PROGRAM PRG_Cycle
VAR	
Status : INT := 0;
bHomingDone: BOOL;
bCycleDone: BOOL;
SFCReset : BOOL;
END_VAR

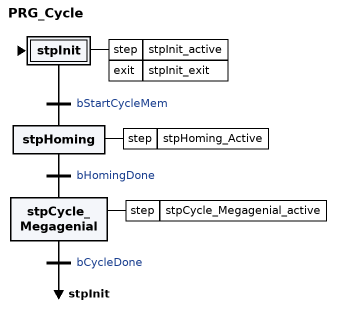
INITIAL_STEP stpInit:
    stpInit_active(N);  // step action
    stpInit_exit(P0);  // exit action
END_STEP
TRANSITION FROM stpInit TO stpHoming
    := bStartCycleMem;
END_TRANSITION
STEP stpHoming:
    stpHoming_Active(N);  // step action
END_STEP
TRANSITION FROM stpHoming TO stpCycle_Megagenial
    := bHomingDone;
END_TRANSITION
STEP stpCycle_Megagenial:
    stpCycle_Megagenial_active(N);  // step action
END_STEP
TRANSITION FROM stpCycle_Megagenial TO stpInit
    := bCycleDone;
END_TRANSITION

ACTION _astpCatch_Rail1_active:
Status := F_IssueActuatorCommand(sDevice := 'R1_Chariot', bArg := TRUE);

CASE Status OF
	1: Result := 0;
	
	0: //Continue
	
	-1: bStopCycleMem := FALSE;
		bStartCycleMem := FALSE;
		bHomingDone := FALSE;
		bCycleDone := FALSE;
		Result := 0;
		SFCReset := TRUE;
END_CASE
END_ACTION

ACTION _astpCatch_Rail1_entry:
Status := 0;
END_ACTION

ACTION _astpCatch_Rail2_active:
Status := F_IssueActuatorCommand(sDevice := 'R2_Chariot', bArg := TRUE);

CASE Status OF
	1: Result := 0;
	
	0: //Continue
	
	-1: bStopCycleMem := FALSE;
		bStartCycleMem := FALSE;
		bHomingDone := FALSE;
		bCycleDone := FALSE;
		Result := 0;
		SFCReset := TRUE;
END_CASE
END_ACTION

ACTION _astpCatch_Rail2_entry:
Status := 0;
END_ACTION

ACTION _astpCatch_Rail3_active:
Status := F_IssueActuatorCommand(sDevice := 'R3_Chariot', bArg := TRUE);

CASE Status OF
	1: Result := 0;
	
	0: //Continue
	
	-1: bStopCycleMem := FALSE;
		bStartCycleMem := FALSE;
		bHomingDone := FALSE;
		bCycleDone := FALSE;
		Result := 0;
		SFCReset := TRUE;
END_CASE
END_ACTION

ACTION _astpCatch_Rail3_entry:
Status := 0;
END_ACTION

ACTION _astpCatch_Rail4_active:
Status := F_IssueActuatorCommand(sDevice := 'R4_Chariot', bArg := TRUE);

CASE Status OF
	1: Result := 0;
	
	0: //Continue
	
	-1: bStopCycleMem := FALSE;
		bStartCycleMem := FALSE;
		bHomingDone := FALSE;
		bCycleDone := FALSE;
		Result := 0;
		SFCReset := TRUE;
END_CASE
END_ACTION

ACTION _astpCatch_Rail4_entry:
Status := 0;
END_ACTION

ACTION _astpCatchPickUp_Rail3_active:
Status := F_IssueActuatorCommand(sDevice := 'R3_Chariot', bArg := TRUE);

CASE Status OF
	1: Result := 0;
	
	0: //Contionue
	
	-1: bStopCycleMem := FALSE;
		bStartCycleMem := FALSE;
		bHomingDone := FALSE;
		bCycleDone := FALSE;
		Result := 0;
		SFCReset := TRUE;
END_CASE
END_ACTION

ACTION _astpCatchPickUp_Rail3_entry:
Status := 0;
END_ACTION

ACTION _astpDrop_Gui1_active:
Status := F_IssueActuatorCommand(sDevice := 'R3_HeatExCoupola', bArg := FALSE);

CASE Status OF
	1: Result := 0;
	
	0: //Continue
	
	-1: bStopCycleMem := FALSE;
		bStartCycleMem := FALSE;
		bHomingDone := FALSE;
		bCycleDone := FALSE;
		Result := 0;
		SFCReset := TRUE;
END_CASE
END_ACTION

ACTION _astpDrop_Gui1_entry:
Status := 0;
END_ACTION

ACTION _astpDrop_Rail1_entry:
Status := 0;
END_ACTION

ACTION _astpDrop_Rail2_active:
Status := F_IssueActuatorCommand(sDevice := 'R2_Chariot', bArg := FALSE);

CASE Status OF
	1: Result := 0;
	
	0: //Continue
	
	-1: bStopCycleMem := FALSE;
		bStartCycleMem := FALSE;
		bHomingDone := FALSE;
		bCycleDone := FALSE;
		Result := 0;
		SFCReset := TRUE;
END_CASE
END_ACTION

ACTION _astpDrop_Rail2_entry:
Status := 0;
END_ACTION

ACTION _astpDrop_Rail3_active:
Status := F_IssueActuatorCommand(sDevice := 'R3_Chariot', bArg := FALSE);

CASE Status OF
	1: Result := 0;
	
	0: //Continue
	
	-1: bStopCycleMem := FALSE;
		bStartCycleMem := FALSE;
		bHomingDone := FALSE;
		bCycleDone := FALSE;
		Result := 0;
		SFCReset := TRUE;
END_CASE
END_ACTION

ACTION _astpDrop_Rail3_entry:
Status := 0;
END_ACTION

ACTION _astpDrop_Rail4_active_1:
Status := F_IssueActuatorCommand(sDevice := 'R4_Chariot', bArg := FALSE);

CASE Status OF
	1: Result := 0;
	
	0: //Continue
	
	-1: bStopCycleMem := FALSE;
		bStartCycleMem := FALSE;
		bHomingDone := FALSE;
		bCycleDone := FALSE;
		Result := 0;
		SFCReset := TRUE;
END_CASE
END_ACTION

ACTION _astpDrop_Rail4_entry:
Status := 0;
END_ACTION

ACTION _astpDropMoveFinal_Rail3_active:
Status := F_IssueActuatorCommand(sDevice := 'R3_Chariot', bArg := FALSE);

CASE Status OF
	1: Result := 0;
	
	0: //Contionue
	
	-1: bStopCycleMem := FALSE;
		bStartCycleMem := FALSE;
		bHomingDone := FALSE;
		bCycleDone := FALSE;
		Result := 0;
		SFCReset := TRUE;
END_CASE
END_ACTION

ACTION _astpDropMoveFinal_Rail3_entry:
Status := 0;
END_ACTION

ACTION _astpEnd_active:
IF bStopCycleMem THEN
	bStartCycleMem := FALSE;
	bStopCycleMem := FALSE;
	bHomingDone := FALSE;
END_IF

bHomingDone := FALSE;
bCycleDone := TRUE;
END_ACTION

ACTION _astpExtend_Pous2_active:
Status := F_IssueActuatorCommand(sDevice := 'R3_Compressor', bArg := TRUE);

CASE Status OF
	1: Result := 0;
	
	0: //Continue
	
	-1: bStopCycleMem := FALSE;
		bStartCycleMem := FALSE;
		bHomingDone := FALSE;
		bCycleDone := FALSE;
		Result := 0;
		SFCReset := TRUE;
END_CASE
END_ACTION

ACTION _astpExtend_Pous2_entry:
Status := 0;
END_ACTION

ACTION _astpHoming_Gui1_active:
Status := F_IssueActuatorCommand(sDevice := 'R3_HeatExCoupola', bArg := TRUE);

CASE Status OF
	1: Result := 0;
	
	0: //Continue
	
	-1: bStopCycleMem := FALSE;
		bStartCycleMem := FALSE;
		bHomingDone := FALSE;
		bCycleDone := FALSE;
		Result := 0;
		SFCReset := TRUE;
END_CASE
END_ACTION

ACTION _astpHoming_Gui1_entry:
Status := 0;
END_ACTION

ACTION _astpHoming_Gui2_active:
Status := F_IssueActuatorCommand(sDevice := 'R3_RegenCoupola', bArg := TRUE);

CASE Status OF
	1: Result := 0;
	
	0: //Continue
	
	-1: bStopCycleMem := FALSE;
		bStartCycleMem := FALSE;
		bHomingDone := FALSE;
		bCycleDone := FALSE;
		Result := 0;
		SFCReset := TRUE;
END_CASE
END_ACTION

ACTION _astpHoming_Gui2_entry:
Status := 0;
END_ACTION

ACTION _astpHoming_Pous1_active:
Status := F_IssueActuatorCommand(sDevice := 'R1_Compressor', bArg := FALSE);

CASE Status OF
	1: Result := 0;
	
	0: //Continue
	
	-1: bStopCycleMem := FALSE;
		bStartCycleMem := FALSE;
		bHomingDone := FALSE;
		bCycleDone := FALSE;
		Result := 0;
		SFCReset := TRUE;
END_CASE
END_ACTION

ACTION _astpHoming_Pous1_entry:
Status := 0;
END_ACTION

ACTION _astpHoming_Pous2_active:
Status := F_IssueActuatorCommand(sDevice := 'R3_Compressor', bArg := FALSE);

CASE Status OF
	1: Result := 0;
	   bHomingDone := TRUE;
	
	0: //Continue
	
	-1: bStopCycleMem := FALSE;
		bStartCycleMem := FALSE;
		bHomingDone := FALSE;
		bCycleDone := FALSE;
		Result := 0;
		SFCReset := TRUE;
END_CASE
END_ACTION

ACTION _astpHoming_Pous2_entry:
Status := 0;
END_ACTION

ACTION _astpHoming_Rail1_entry:
Status := 0;
END_ACTION

ACTION _astpHoming_Rail2_entry:
Status := 0;
END_ACTION

ACTION _astpHoming_Rail3_entry:
Status := 0;
END_ACTION

ACTION _astpHoming_Rail4_entry:
Status := 0;
END_ACTION

ACTION _astpHoming_Tri1_active:
Status := F_IssueActuatorCommand(sDevice := 'R1_Chariot', bArg := FALSE);

CASE Status OF
	1: Result := 0;
	
	0: //Continue
	
	-1: bStopCycleMem := FALSE;
		bStartCycleMem := FALSE;
		bHomingDone := FALSE;
		bCycleDone := FALSE;
		Result := 0;
		SFCReset := TRUE;
END_CASE
END_ACTION

ACTION _astpHoming_Tri1_entry:
Status := 0;
END_ACTION

ACTION _astpHoming_Tri2_active:
IF bStopCycleMem THEN
	sRequestedActuator := 'none';
	CancelMove := TRUE;
ELSIF NOT bStopCycleMem THEN
	Status := F_IssueActuatorCommand(sDevice := 'R2_Chariot', bArg := FALSE);
END_IF

IF Status = 1 THEN
	Result := 0;
END_IF
END_ACTION

ACTION _astpHoming_Tri2_active_1:
Status := F_IssueActuatorCommand(sDevice := 'R2_Chariot', bArg := FALSE);

CASE Status OF
	1: Result := 0;
	
	0: //Continue
	
	-1: bStopCycleMem := FALSE;
		bStartCycleMem := FALSE;
		bHomingDone := FALSE;
		bCycleDone := FALSE;
		Result := 0;
		SFCReset := TRUE;
END_CASE
END_ACTION

ACTION _astpHoming_Tri2_entry:
Status := 0;
END_ACTION

ACTION _astpHoming_Tri2_entry_1:
Status := 0;
END_ACTION

ACTION _astpHoming_Tri3_active:
Status := F_IssueActuatorCommand(sDevice := 'R3_Chariot', bArg := FALSE);

CASE Status OF
	1: Result := 0;
	
	0: //Continue
	
	-1: bStopCycleMem := FALSE;
		bStartCycleMem := FALSE;
		bHomingDone := FALSE;
		bCycleDone := FALSE;
		Result := 0;
		SFCReset := TRUE;
END_CASE
END_ACTION

ACTION _astpHoming_Tri3_entry:
Status := 0;
END_ACTION

ACTION _astpHoming_Tri4_active:
Status := F_IssueActuatorCommand(sDevice := 'R4_Chariot', bArg := FALSE);

CASE Status OF
	1: Result := 0;
	
	0: //Continue
	
	-1: bStopCycleMem := FALSE;
		bStartCycleMem := FALSE;
		bHomingDone := FALSE;
		bCycleDone := FALSE;
		Result := 0;
		SFCReset := TRUE;
END_CASE
END_ACTION

ACTION _astpHoming_Tri4_entry:
Status := 0;
END_ACTION

ACTION _astpInit_Cycle_Megagenial_active:

END_ACTION

ACTION _astpInit_Homing_active:

END_ACTION

ACTION _astpMoveBw_Rail1_active:
Status := F_IssueActuatorCommand(sDevice := 'R1_Motor', bArg := FALSE, bHasPosition := TRUE, nPosition:= 6, fVelocity := Mot_LoadedVel);
	
CASE Status OF
	1: Result := 0;
	
	0: //Continue
	
	-1: bStopCycleMem := FALSE;
		bStartCycleMem := FALSE;
		bHomingDone := FALSE;
		bCycleDone := FALSE;
		Result := 0;
		SFCReset := TRUE;
END_CASE
END_ACTION

ACTION _astpMoveBw_Rail1_entry:
Status := 0;
END_ACTION

ACTION _astpMoveBw_Rail2_active:
Status := F_IssueActuatorCommand(sDevice := 'R2_Motor', bArg := FALSE, bHasPosition := TRUE, nPosition:= 6, fVelocity := Mot_LoadedVel);

CASE Status OF
	1: Result := 0;
	
	0: //Continue
	
	-1: bStopCycleMem := FALSE;
		bStartCycleMem := FALSE;
		bHomingDone := FALSE;
		bCycleDone := FALSE;
		Result := 0;
		SFCReset := TRUE;
END_CASE
END_ACTION

ACTION _astpMoveBw_Rail2_entry:
Status := 0;
END_ACTION

ACTION _astpMoveBw_Rail3_active:
Status := F_IssueActuatorCommand(sDevice := 'R3_Motor', bArg := FALSE, bHasPosition := TRUE, nPosition:= 6, fVelocity := Mot_LoadedVel);
	
CASE Status OF
	1: Result := 0;
	
	0: //Continue
	
	-1: bStopCycleMem := FALSE;
		bStartCycleMem := FALSE;
		bHomingDone := FALSE;
		bCycleDone := FALSE;
		Result := 0;
		SFCReset := TRUE;
END_CASE
END_ACTION

ACTION _astpMoveBw_Rail3_entry:
Status := 0;
END_ACTION

ACTION _astpMoveBw_Rail4_active:
Status := F_IssueActuatorCommand(sDevice := 'R4_Motor', bArg := FALSE, bHasPosition := TRUE, nPosition:= 9, fVelocity := Mot_LoadedVel);

CASE Status OF
	1: Result := 0;
	
	0: //Continue
	
	-1: bStopCycleMem := FALSE;
		bStartCycleMem := FALSE;
		bHomingDone := FALSE;
		bCycleDone := FALSE;
		Result := 0;
		SFCReset := TRUE;
END_CASE
END_ACTION

ACTION _astpMoveBw_Rail4_entry:
Status := 0;
END_ACTION

ACTION _astpMoveFinal_Rail3_active:
Status := F_IssueActuatorCommand(sDevice := 'R3_Motor', bArg := FALSE, bHasPosition := TRUE, nPosition:= 6, fVelocity := Mot_UnloadedVel);

CASE Status OF
	1: Result := 0;
	
	0: //Contionue
	
	-1: bStopCycleMem := FALSE;
		bStartCycleMem := FALSE;
		bHomingDone := FALSE;
		bCycleDone := FALSE;
		Result := 0;
		SFCReset := TRUE;
END_CASE
END_ACTION

ACTION _astpMoveFinal_Rail3_entry:
Status := 0;
END_ACTION

ACTION _astpMoveFw_Rail1_active:
Status := F_IssueActuatorCommand(sDevice := 'R1_Motor', bArg := FALSE, bHasPosition := TRUE, nPosition:= 1290, fVelocity := Mot_UnloadedVel);

CASE Status OF
	1: Result := 0;
	
	0: //Continue
	
	-1: bStopCycleMem := FALSE;
		bStartCycleMem := FALSE;
		bHomingDone := FALSE;
		bCycleDone := FALSE;
		Result := 0;
		SFCReset := TRUE;
END_CASE
END_ACTION

ACTION _astpMoveFw_Rail1_entry:
Status := 0;
END_ACTION

ACTION _astpMoveFw_Rail2_active:
Status := F_IssueActuatorCommand(sDevice := 'R2_Motor', bArg := FALSE, bHasPosition := TRUE, nPosition:= 980, fVelocity := Mot_UnloadedVel);

CASE Status OF
	1: Result := 0;
	
	0: //Continue
	
	-1: bStopCycleMem := FALSE;
		bStartCycleMem := FALSE;
		bHomingDone := FALSE;
		bCycleDone := FALSE;
		Result := 0;
		SFCReset := TRUE;
END_CASE
END_ACTION

ACTION _astpMoveFw_Rail2_entry:
Status := 0;
END_ACTION

ACTION _astpMoveFw_Rail3_active:
Status := F_IssueActuatorCommand(sDevice := 'R3_Motor', bArg := FALSE, bHasPosition := TRUE, nPosition:= 1290, fVelocity := Mot_UnloadedVel);

CASE Status OF
	1: Result := 0;
	
	0: //Contionue
	
	-1: bStopCycleMem := FALSE;
		bStartCycleMem := FALSE;
		bHomingDone := FALSE;
		bCycleDone := FALSE;
		Result := 0;
		SFCReset := TRUE;
END_CASE
END_ACTION

ACTION _astpMoveFw_Rail3_entry:
Status := 0;
END_ACTION

ACTION _astpMoveFw_Rail4_active:
Status := F_IssueActuatorCommand(sDevice := 'R4_Motor', bArg := FALSE, bHasPosition := TRUE, nPosition:= 980, fVelocity := Mot_UnloadedVel);

CASE Status OF
	1: Result := 0;
	
	0: //Continue
	
	-1: bStopCycleMem := FALSE;
		bStartCycleMem := FALSE;
		bHomingDone := FALSE;
		bCycleDone := FALSE;
		Result := 0;
		SFCReset := TRUE;
END_CASE
END_ACTION

ACTION _astpMoveFw_Rail4_entry:
Status := 0;
END_ACTION

ACTION _astpMovePickUp_Rail3_active:
Status := F_IssueActuatorCommand(sDevice := 'R3_Motor', bArg := FALSE, bHasPosition := TRUE, nPosition:= 150, fVelocity := Mot_UnloadedVel);

CASE Status OF
	1: Result := 0;
	
	0: //Contionue
	
	-1: bStopCycleMem := FALSE;
		bStartCycleMem := FALSE;
		bHomingDone := FALSE;
		bCycleDone := FALSE;
		Result := 0;
		SFCReset := TRUE;
END_CASE
END_ACTION

ACTION _astpMovePickUp_Rail3_entry:
Status := 0;
END_ACTION

ACTION _astpPivotIn_active:
Status := F_IssueActuatorCommand(sDevice := 'R1_Sensor', bArg := FALSE);

CASE Status OF
	1: Result := 0;
	
	0: //Continue
	
	-1: bStopCycleMem := FALSE;
		bStartCycleMem := FALSE;
		bHomingDone := FALSE;
		bCycleDone := FALSE;
		Result := 0;
		SFCReset := TRUE;
END_CASE
END_ACTION

ACTION _astpPivotIn_entry:
Status := 0;
END_ACTION

ACTION _astpPivotOut_active:
Status := F_IssueActuatorCommand(sDevice := 'R1_Sensor', bArg := TRUE);

CASE Status OF
	1: Result := 0;
	
	0: //Continue
	
	-1: bStopCycleMem := FALSE;
		bStartCycleMem := FALSE;
		bHomingDone := FALSE;
		bCycleDone := FALSE;
		Result := 0;
		SFCReset := TRUE;
END_CASE
END_ACTION

ACTION _astpPivotOut_entry:
Status := 0;
END_ACTION

ACTION _astpRetract_Gui1_active:
Status := F_IssueActuatorCommand(sDevice := 'R3_HeatExCoupola', bArg := TRUE);

CASE Status OF
	1: Result := 0;
	
	0: //Contionue
	
	-1: bStopCycleMem := FALSE;
		bStartCycleMem := FALSE;
		bHomingDone := FALSE;
		bCycleDone := FALSE;
		Result := 0;
		SFCReset := TRUE;
END_CASE
END_ACTION

ACTION _astpRetract_Gui1_entry:
Status := 0;
END_ACTION

ACTION _astpRetract_Pous2_active:
Status := F_IssueActuatorCommand(sDevice := 'R3_Compressor', bArg := FALSE);

CASE Status OF
	1: Result := 0;
	
	0: //Continue
	
	-1: bStopCycleMem := FALSE;
		bStartCycleMem := FALSE;
		bHomingDone := FALSE;
		bCycleDone := FALSE;
		Result := 0;
		SFCReset := TRUE;
END_CASE
END_ACTION

ACTION _astpRetract_Pous2_entry:
Status := 0;
END_ACTION

ACTION stpCycle_Megagenial_active:
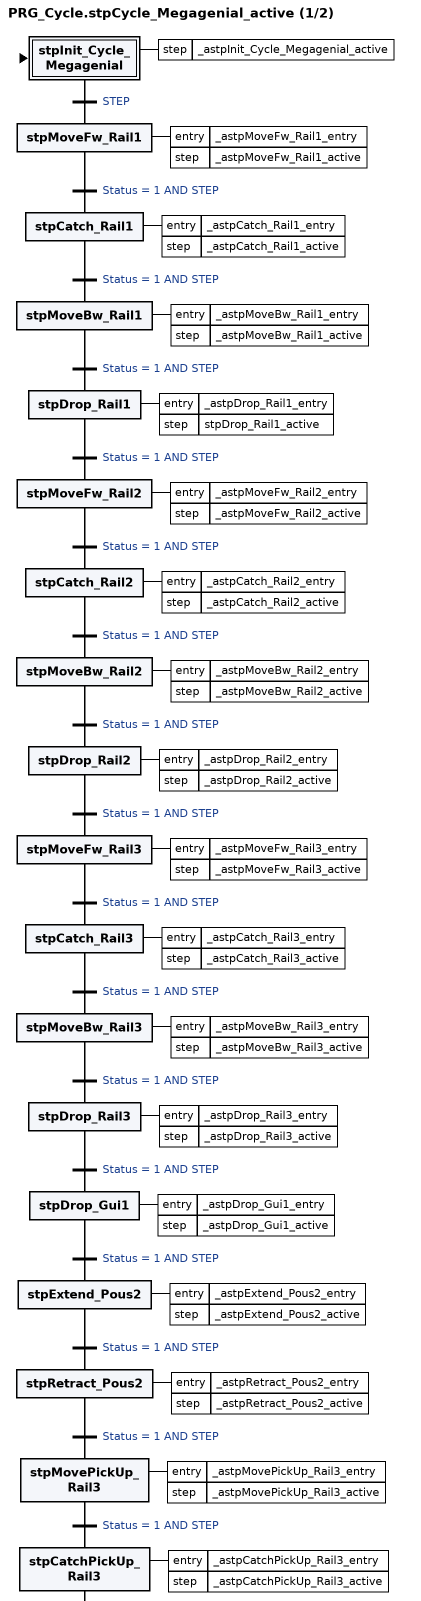
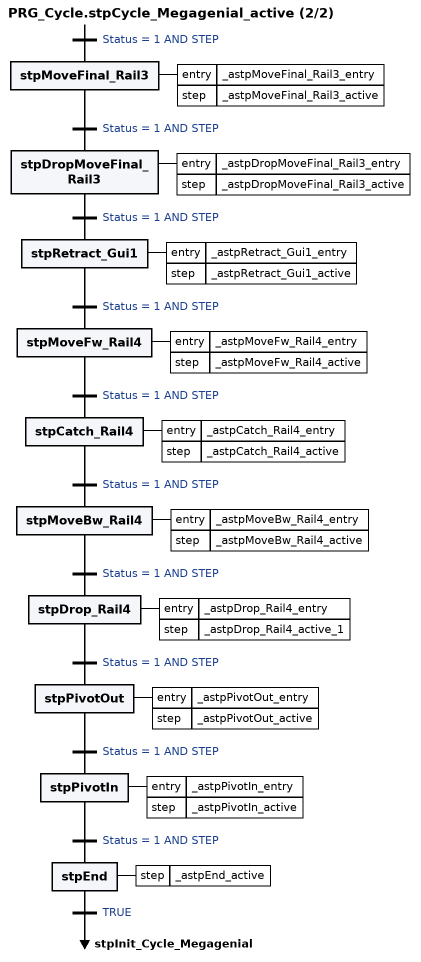
INITIAL_STEP stpInit_Cycle_Megagenial:
    _astpInit_Cycle_Megagenial_active(N);  // step action
END_STEP
TRANSITION FROM stpInit_Cycle_Megagenial TO stpMoveFw_Rail1
    := STEP;
END_TRANSITION
STEP stpMoveFw_Rail1:
    _astpMoveFw_Rail1_entry(P1);  // entry action
    _astpMoveFw_Rail1_active(N);  // step action
END_STEP
TRANSITION FROM stpMoveFw_Rail1 TO stpCatch_Rail1
    := Status = 1 AND STEP;
END_TRANSITION
STEP stpCatch_Rail1:
    _astpCatch_Rail1_entry(P1);  // entry action
    _astpCatch_Rail1_active(N);  // step action
END_STEP
TRANSITION FROM stpCatch_Rail1 TO stpMoveBw_Rail1
    := Status = 1 AND STEP;
END_TRANSITION
STEP stpMoveBw_Rail1:
    _astpMoveBw_Rail1_entry(P1);  // entry action
    _astpMoveBw_Rail1_active(N);  // step action
END_STEP
TRANSITION FROM stpMoveBw_Rail1 TO stpDrop_Rail1
    := Status = 1 AND STEP;
END_TRANSITION
STEP stpDrop_Rail1:
    _astpDrop_Rail1_entry(P1);  // entry action
    stpDrop_Rail1_active(N);  // step action
END_STEP
TRANSITION FROM stpDrop_Rail1 TO stpMoveFw_Rail2
    := Status = 1 AND STEP;
END_TRANSITION
STEP stpMoveFw_Rail2:
    _astpMoveFw_Rail2_entry(P1);  // entry action
    _astpMoveFw_Rail2_active(N);  // step action
END_STEP
TRANSITION FROM stpMoveFw_Rail2 TO stpCatch_Rail2
    := Status = 1 AND STEP;
END_TRANSITION
STEP stpCatch_Rail2:
    _astpCatch_Rail2_entry(P1);  // entry action
    _astpCatch_Rail2_active(N);  // step action
END_STEP
TRANSITION FROM stpCatch_Rail2 TO stpMoveBw_Rail2
    := Status = 1 AND STEP;
END_TRANSITION
STEP stpMoveBw_Rail2:
    _astpMoveBw_Rail2_entry(P1);  // entry action
    _astpMoveBw_Rail2_active(N);  // step action
END_STEP
TRANSITION FROM stpMoveBw_Rail2 TO stpDrop_Rail2
    := Status = 1 AND STEP;
END_TRANSITION
STEP stpDrop_Rail2:
    _astpDrop_Rail2_entry(P1);  // entry action
    _astpDrop_Rail2_active(N);  // step action
END_STEP
TRANSITION FROM stpDrop_Rail2 TO stpMoveFw_Rail3
    := Status = 1 AND STEP;
END_TRANSITION
STEP stpMoveFw_Rail3:
    _astpMoveFw_Rail3_entry(P1);  // entry action
    _astpMoveFw_Rail3_active(N);  // step action
END_STEP
TRANSITION FROM stpMoveFw_Rail3 TO stpCatch_Rail3
    := Status = 1 AND STEP;
END_TRANSITION
STEP stpCatch_Rail3:
    _astpCatch_Rail3_entry(P1);  // entry action
    _astpCatch_Rail3_active(N);  // step action
END_STEP
TRANSITION FROM stpCatch_Rail3 TO stpMoveBw_Rail3
    := Status = 1 AND STEP;
END_TRANSITION
STEP stpMoveBw_Rail3:
    _astpMoveBw_Rail3_entry(P1);  // entry action
    _astpMoveBw_Rail3_active(N);  // step action
END_STEP
TRANSITION FROM stpMoveBw_Rail3 TO stpDrop_Rail3
    := Status = 1 AND STEP;
END_TRANSITION
STEP stpDrop_Rail3:
    _astpDrop_Rail3_entry(P1);  // entry action
    _astpDrop_Rail3_active(N);  // step action
END_STEP
TRANSITION FROM stpDrop_Rail3 TO stpDrop_Gui1
    := Status = 1 AND STEP;
END_TRANSITION
STEP stpDrop_Gui1:
    _astpDrop_Gui1_entry(P1);  // entry action
    _astpDrop_Gui1_active(N);  // step action
END_STEP
TRANSITION FROM stpDrop_Gui1 TO stpExtend_Pous2
    := Status = 1 AND STEP;
END_TRANSITION
STEP stpExtend_Pous2:
    _astpExtend_Pous2_entry(P1);  // entry action
    _astpExtend_Pous2_active(N);  // step action
END_STEP
TRANSITION FROM stpExtend_Pous2 TO stpRetract_Pous2
    := Status = 1 AND STEP;
END_TRANSITION
STEP stpRetract_Pous2:
    _astpRetract_Pous2_entry(P1);  // entry action
    _astpRetract_Pous2_active(N);  // step action
END_STEP
TRANSITION FROM stpRetract_Pous2 TO stpMovePickUp_Rail3
    := Status = 1 AND STEP;
END_TRANSITION
STEP stpMovePickUp_Rail3:
    _astpMovePickUp_Rail3_entry(P1);  // entry action
    _astpMovePickUp_Rail3_active(N);  // step action
END_STEP
TRANSITION FROM stpMovePickUp_Rail3 TO stpCatchPickUp_Rail3
    := Status = 1 AND STEP;
END_TRANSITION
STEP stpCatchPickUp_Rail3:
    _astpCatchPickUp_Rail3_entry(P1);  // entry action
    _astpCatchPickUp_Rail3_active(N);  // step action
END_STEP
TRANSITION FROM stpCatchPickUp_Rail3 TO stpMoveFinal_Rail3
    := Status = 1 AND STEP;
END_TRANSITION
STEP stpMoveFinal_Rail3:
    _astpMoveFinal_Rail3_entry(P1);  // entry action
    _astpMoveFinal_Rail3_active(N);  // step action
END_STEP
TRANSITION FROM stpMoveFinal_Rail3 TO stpDropMoveFinal_Rail3
    := Status = 1 AND STEP;
END_TRANSITION
STEP stpDropMoveFinal_Rail3:
    _astpDropMoveFinal_Rail3_entry(P1);  // entry action
    _astpDropMoveFinal_Rail3_active(N);  // step action
END_STEP
TRANSITION FROM stpDropMoveFinal_Rail3 TO stpRetract_Gui1
    := Status = 1 AND STEP;
END_TRANSITION
STEP stpRetract_Gui1:
    _astpRetract_Gui1_entry(P1);  // entry action
    _astpRetract_Gui1_active(N);  // step action
END_STEP
TRANSITION FROM stpRetract_Gui1 TO stpMoveFw_Rail4
    := Status = 1 AND STEP;
END_TRANSITION
STEP stpMoveFw_Rail4:
    _astpMoveFw_Rail4_entry(P1);  // entry action
    _astpMoveFw_Rail4_active(N);  // step action
END_STEP
TRANSITION FROM stpMoveFw_Rail4 TO stpCatch_Rail4
    := Status = 1 AND STEP;
END_TRANSITION
STEP stpCatch_Rail4:
    _astpCatch_Rail4_entry(P1);  // entry action
    _astpCatch_Rail4_active(N);  // step action
END_STEP
TRANSITION FROM stpCatch_Rail4 TO stpMoveBw_Rail4
    := Status = 1 AND STEP;
END_TRANSITION
STEP stpMoveBw_Rail4:
    _astpMoveBw_Rail4_entry(P1);  // entry action
    _astpMoveBw_Rail4_active(N);  // step action
END_STEP
TRANSITION FROM stpMoveBw_Rail4 TO stpDrop_Rail4
    := Status = 1 AND STEP;
END_TRANSITION
STEP stpDrop_Rail4:
    _astpDrop_Rail4_entry(P1);  // entry action
    _astpDrop_Rail4_active_1(N);  // step action
END_STEP
TRANSITION FROM stpDrop_Rail4 TO stpPivotOut
    := Status = 1 AND STEP;
END_TRANSITION
STEP stpPivotOut:
    _astpPivotOut_entry(P1);  // entry action
    _astpPivotOut_active(N);  // step action
END_STEP
TRANSITION FROM stpPivotOut TO stpPivotIn
    := Status = 1 AND STEP;
END_TRANSITION
STEP stpPivotIn:
    _astpPivotIn_entry(P1);  // entry action
    _astpPivotIn_active(N);  // step action
END_STEP
TRANSITION FROM stpPivotIn TO stpEnd
    := Status = 1 AND STEP;
END_TRANSITION
STEP stpEnd:
    _astpEnd_active(N);  // step action
END_STEP
TRANSITION FROM stpEnd TO stpInit_Cycle_Megagenial
    := TRUE;
END_TRANSITION
END_ACTION

ACTION stpDrop_Rail1_active:
Status := F_IssueActuatorCommand(sDevice := 'R1_Chariot', bArg := FALSE);
 
CASE Status OF
	1: Result := 0;
	
	0: //Continue
	
	-1: bStopCycleMem := FALSE;
		bStartCycleMem := FALSE;
		bHomingDone := FALSE;
		bCycleDone := FALSE;
		Result := 0;
		SFCReset := TRUE;
END_CASE
END_ACTION

ACTION stpHoming_Active:
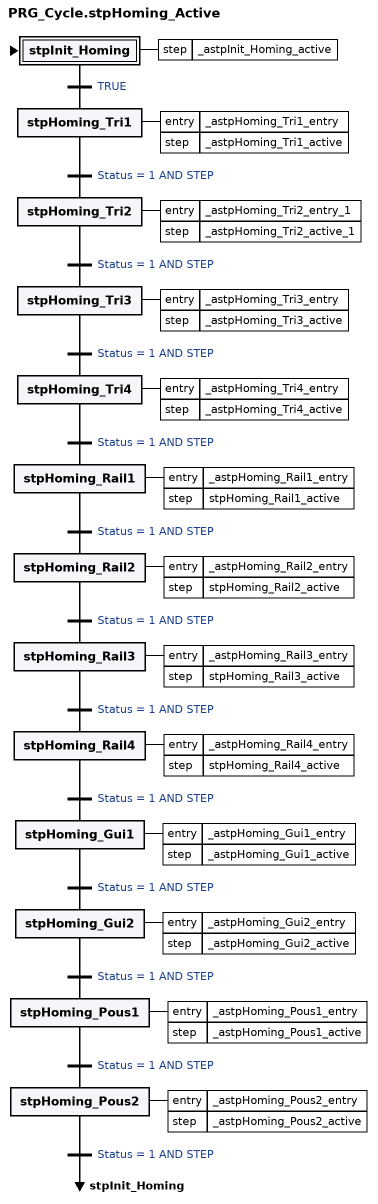
INITIAL_STEP stpInit_Homing:
    _astpInit_Homing_active(N);  // step action
END_STEP
TRANSITION FROM stpInit_Homing TO stpHoming_Tri1
    := TRUE;
END_TRANSITION
STEP stpHoming_Tri1:
    _astpHoming_Tri1_entry(P1);  // entry action
    _astpHoming_Tri1_active(N);  // step action
END_STEP
TRANSITION FROM stpHoming_Tri1 TO stpHoming_Tri2
    := Status = 1 AND STEP;
END_TRANSITION
STEP stpHoming_Tri2:
    _astpHoming_Tri2_entry_1(P1);  // entry action
    _astpHoming_Tri2_active_1(N);  // step action
END_STEP
TRANSITION FROM stpHoming_Tri2 TO stpHoming_Tri3
    := Status = 1 AND STEP;
END_TRANSITION
STEP stpHoming_Tri3:
    _astpHoming_Tri3_entry(P1);  // entry action
    _astpHoming_Tri3_active(N);  // step action
END_STEP
TRANSITION FROM stpHoming_Tri3 TO stpHoming_Tri4
    := Status = 1 AND STEP;
END_TRANSITION
STEP stpHoming_Tri4:
    _astpHoming_Tri4_entry(P1);  // entry action
    _astpHoming_Tri4_active(N);  // step action
END_STEP
TRANSITION FROM stpHoming_Tri4 TO stpHoming_Rail1
    := Status = 1 AND STEP;
END_TRANSITION
STEP stpHoming_Rail1:
    _astpHoming_Rail1_entry(P1);  // entry action
    stpHoming_Rail1_active(N);  // step action
END_STEP
TRANSITION FROM stpHoming_Rail1 TO stpHoming_Rail2
    := Status = 1 AND STEP;
END_TRANSITION
STEP stpHoming_Rail2:
    _astpHoming_Rail2_entry(P1);  // entry action
    stpHoming_Rail2_active(N);  // step action
END_STEP
TRANSITION FROM stpHoming_Rail2 TO stpHoming_Rail3
    := Status = 1 AND STEP;
END_TRANSITION
STEP stpHoming_Rail3:
    _astpHoming_Rail3_entry(P1);  // entry action
    stpHoming_Rail3_active(N);  // step action
END_STEP
TRANSITION FROM stpHoming_Rail3 TO stpHoming_Rail4
    := Status = 1 AND STEP;
END_TRANSITION
STEP stpHoming_Rail4:
    _astpHoming_Rail4_entry(P1);  // entry action
    stpHoming_Rail4_active(N);  // step action
END_STEP
TRANSITION FROM stpHoming_Rail4 TO stpHoming_Gui1
    := Status = 1 AND STEP;
END_TRANSITION
STEP stpHoming_Gui1:
    _astpHoming_Gui1_entry(P1);  // entry action
    _astpHoming_Gui1_active(N);  // step action
END_STEP
TRANSITION FROM stpHoming_Gui1 TO stpHoming_Gui2
    := Status = 1 AND STEP;
END_TRANSITION
STEP stpHoming_Gui2:
    _astpHoming_Gui2_entry(P1);  // entry action
    _astpHoming_Gui2_active(N);  // step action
END_STEP
TRANSITION FROM stpHoming_Gui2 TO stpHoming_Pous1
    := Status = 1 AND STEP;
END_TRANSITION
STEP stpHoming_Pous1:
    _astpHoming_Pous1_entry(P1);  // entry action
    _astpHoming_Pous1_active(N);  // step action
END_STEP
TRANSITION FROM stpHoming_Pous1 TO stpHoming_Pous2
    := Status = 1 AND STEP;
END_TRANSITION
STEP stpHoming_Pous2:
    _astpHoming_Pous2_entry(P1);  // entry action
    _astpHoming_Pous2_active(N);  // step action
END_STEP
TRANSITION FROM stpHoming_Pous2 TO stpInit_Homing
    := Status = 1 AND STEP;
END_TRANSITION
END_ACTION

ACTION stpHoming_Rail1_active:
Status := F_IssueActuatorCommand(sDevice := 'R1_Motor', bArg := TRUE);

CASE Status OF
	1: Result := 0;
	
	0: //Continue
	
	-1: bStopCycleMem := FALSE;
		bStartCycleMem := FALSE;
		bHomingDone := FALSE;
		bCycleDone := FALSE;
		Result := 0;
		SFCReset := TRUE;
END_CASE
END_ACTION

ACTION stpHoming_Rail2_active:
Status := F_IssueActuatorCommand(sDevice := 'R2_Motor', bArg := TRUE);

CASE Status OF
	1: Result := 0;
	
	0: //Continue
	
	-1: bStopCycleMem := FALSE;
		bStartCycleMem := FALSE;
		bHomingDone := FALSE;
		bCycleDone := FALSE;
		Result := 0;
		SFCReset := TRUE;
END_CASE
END_ACTION

ACTION stpHoming_Rail3_active:
Status := F_IssueActuatorCommand(sDevice := 'R3_Motor', bArg := TRUE);

CASE Status OF
	1: Result := 0;
	
	0: //Continue
	
	-1: bStopCycleMem := FALSE;
		bStartCycleMem := FALSE;
		bHomingDone := FALSE;
		bCycleDone := FALSE;
		Result := 0;
		SFCReset := TRUE;
END_CASE
END_ACTION

ACTION stpHoming_Rail4_active:
Status := F_IssueActuatorCommand(sDevice := 'R4_Motor', bArg := TRUE);

CASE Status OF
	1: Result := 0;
	
	0: //Continue
	
	-1: bStopCycleMem := FALSE;
		bStartCycleMem := FALSE;
		bHomingDone := FALSE;
		bCycleDone := FALSE;
		Result := 0;
		SFCReset := TRUE;
END_CASE
END_ACTION

ACTION stpInit_active:
SFCReset := FALSE;

(* Read Inputs *)
RTrigStart(CLK := StartCycle OR StartCycle_HMI);
RTrigStop (CLK := StopCycle OR StopCycle_HMI);

IF RTrigStart.Q THEN
    bStartCycleMem := TRUE;   
    StartCycle_HMI := FALSE; 
END_IF

IF RTrigStop.Q THEN
    bStopCycleMem  := TRUE;
    StopCycle_HMI := FALSE;
END_IF
END_ACTION

ACTION stpInit_exit:
bCycleDone := FALSE;
Result := 0;
END_ACTION

END_PROGRAM

(* stored: Version 1.1.0.1, ProductVersion 3.1.4026.11
   POU PRG_Cycle: Id {944d4077-7520-43a4-9286-0335fef2c8f2}, SpecialFunc None
   Action _astpCatch_Rail1_active: Id {15e5e688-c41d-4e1b-83a4-4a0418a7668f}
   Action _astpCatch_Rail1_entry: Id {bdfde7bc-628f-4a08-90eb-953031ec4601}
   Action _astpCatch_Rail2_active: Id {36e7623b-38d9-43a8-b4dd-60a992f6d719}
   Action _astpCatch_Rail2_entry: Id {274a5ad7-af56-4c9c-b2dc-3617c4b28a6d}
   Action _astpCatch_Rail3_active: Id {f30aa1a2-76d1-4ac1-82e9-5d15aa2bf496}
   Action _astpCatch_Rail3_entry: Id {6189bb92-dd3f-41fa-9442-1e62813196af}
   Action _astpCatch_Rail4_active: Id {97b968df-9c31-4b5b-bf55-b814b8a8efdf}
   Action _astpCatch_Rail4_entry: Id {f6a359cc-ad6a-4a57-aa92-a563aabb4c9f}
   Action _astpCatchPickUp_Rail3_active: Id {dce354aa-cabc-4a4f-a8f8-6976f8e11d6b}
   Action _astpCatchPickUp_Rail3_entry: Id {8def0c7b-4b95-4ad1-ad85-a834704e5906}
   Action _astpDrop_Gui1_active: Id {aca502e7-e91e-493e-803f-ef08dc0df054}
   Action _astpDrop_Gui1_entry: Id {6103af35-1250-4790-a869-5eb00d778ca5}
   Action _astpDrop_Rail1_entry: Id {dd7866e6-0c2a-4c71-9ccc-fc077edbd165}
   Action _astpDrop_Rail2_active: Id {2d4e5bf1-06e4-4a49-84d6-26c0c11f7ba6}
   Action _astpDrop_Rail2_entry: Id {3219babe-58a5-464b-ad1e-ce504d3b3b15}
   Action _astpDrop_Rail3_active: Id {bd9e0576-c9bb-47e1-ae3f-98e11da58804}
   Action _astpDrop_Rail3_entry: Id {76bb0c11-7930-4ab7-a2a0-2b69127bfe3f}
   Action _astpDrop_Rail4_active_1: Id {6663ac16-3028-43c7-82d1-5e8cc51f5ec8}
   Action _astpDrop_Rail4_entry: Id {72fa19a7-d20c-4352-97d0-cad15de129d4}
   Action _astpDropMoveFinal_Rail3_active: Id {c3366381-bb3e-4795-a185-bed895edcb49}
   Action _astpDropMoveFinal_Rail3_entry: Id {e0bd2f9d-3435-445d-999d-d43765e22e0c}
   Action _astpEnd_active: Id {dc4dd89e-03eb-4f8f-9127-19947884d0c5}
   Action _astpExtend_Pous2_active: Id {cd6c919c-30dc-46ec-9a71-5584a9815820}
   Action _astpExtend_Pous2_entry: Id {4f1521a6-2640-413a-85c7-5229eaf09abe}
   Action _astpHoming_Gui1_active: Id {eea42098-7e11-449b-9e3c-1c5d002e8c94}
   Action _astpHoming_Gui1_entry: Id {8d7344fe-2a6f-4865-9650-48e5e336e48e}
   Action _astpHoming_Gui2_active: Id {fe375883-eb9a-4d15-afc8-7aa8543450b8}
   Action _astpHoming_Gui2_entry: Id {54590f6c-729b-4f48-b277-b7f454b92c5b}
   Action _astpHoming_Pous1_active: Id {75730ea4-7107-4c35-9681-08dcb362ce0e}
   Action _astpHoming_Pous1_entry: Id {4b44316a-d849-46eb-b00f-33a978d09f15}
   Action _astpHoming_Pous2_active: Id {62ba4e48-037d-4c24-85fb-b51ef8c16e96}
   Action _astpHoming_Pous2_entry: Id {2d9270e8-239b-4009-b957-964e4dcf5d03}
   Action _astpHoming_Rail1_entry: Id {7e053e09-4ef0-4b89-bd47-d44432589724}
   Action _astpHoming_Rail2_entry: Id {325c9c0c-8a71-4fa6-91c3-19a3f35afeef}
   Action _astpHoming_Rail3_entry: Id {bf459a70-bde3-4a09-b414-45eebfc802a0}
   Action _astpHoming_Rail4_entry: Id {a399ef9d-5bbc-449b-90bf-50e2ec4fd1f0}
   Action _astpHoming_Tri1_active: Id {d48613fc-0cff-4667-862e-e958ad0507f2}
   Action _astpHoming_Tri1_entry: Id {80d01037-dfaa-466a-8988-a5f6554ada59}
   Action _astpHoming_Tri2_active: Id {c04d3f22-a0e4-4630-b19b-b107fd2fd0d1}
   Action _astpHoming_Tri2_active_1: Id {b6a8400f-75e0-4b47-9b29-3fa47fd0503e}
   Action _astpHoming_Tri2_entry: Id {77b0d538-b88a-42bb-8392-3729054c840b}
   Action _astpHoming_Tri2_entry_1: Id {b7e33d8a-8ebe-4298-a2b5-daab9f7b99d8}
   Action _astpHoming_Tri3_active: Id {971962bb-2f64-4d7c-a7be-208fa82164fb}
   Action _astpHoming_Tri3_entry: Id {3ff2b6d8-0782-4496-9a39-e8631377378a}
   Action _astpHoming_Tri4_active: Id {4cb91600-7140-40c9-9842-1156876d3fa0}
   Action _astpHoming_Tri4_entry: Id {4367386c-c132-44ed-9fee-7008d2885b97}
   Action _astpInit_Cycle_Megagenial_active: Id {614323da-31e7-4d4b-b52b-3e0a024f70e3}
   Action _astpInit_Homing_active: Id {309757e9-73b6-42d8-9a1a-85df415823f8}
   Action _astpMoveBw_Rail1_active: Id {82951208-c126-4f3b-b86c-8ccca38af486}
   Action _astpMoveBw_Rail1_entry: Id {3eebb312-5460-4038-8d09-7613c4c13b19}
   Action _astpMoveBw_Rail2_active: Id {8ce7cc61-da1e-4a34-85f2-211cd14887ac}
   Action _astpMoveBw_Rail2_entry: Id {dce9cf22-f69e-476d-96b0-4263aae25079}
   Action _astpMoveBw_Rail3_active: Id {259ee54a-14e3-4e6c-b91e-ad337126d969}
   Action _astpMoveBw_Rail3_entry: Id {13d33900-a017-4f19-a30c-fdb048e6ed6f}
   Action _astpMoveBw_Rail4_active: Id {41541f05-84bc-42f6-ba00-975ac632aeaa}
   Action _astpMoveBw_Rail4_entry: Id {7869959f-1ba7-4e34-9979-54c0cb5859b0}
   Action _astpMoveFinal_Rail3_active: Id {868d3b76-a02b-4e70-8735-9182079229e3}
   Action _astpMoveFinal_Rail3_entry: Id {0ad41103-df29-4c26-9888-9d57b7b88895}
   Action _astpMoveFw_Rail1_active: Id {06e8ca90-ee36-400c-a2c7-f6476c6539a8}
   Action _astpMoveFw_Rail1_entry: Id {a7c0ca7c-1904-4b59-b8cf-622e2a7a6f74}
   Action _astpMoveFw_Rail2_active: Id {2761dac4-bb6c-4875-90ff-e278d49dd75b}
   Action _astpMoveFw_Rail2_entry: Id {e0bc69ca-4003-4fce-90eb-6635978800b2}
   Action _astpMoveFw_Rail3_active: Id {6a96c489-a3a3-4b96-b95c-0c4d2ef3b7d6}
   Action _astpMoveFw_Rail3_entry: Id {9a8d21b1-9e69-47fa-9c44-410eb5d015b1}
   Action _astpMoveFw_Rail4_active: Id {c102d237-2a20-4c62-a356-1f4e48751a2c}
   Action _astpMoveFw_Rail4_entry: Id {44961982-540a-4ab7-9c0a-6bb5f0501515}
   Action _astpMovePickUp_Rail3_active: Id {0bfac081-6762-49da-97b8-c44aba5cf64f}
   Action _astpMovePickUp_Rail3_entry: Id {81d71aa3-7201-45ae-ba83-2224433b5170}
   Action _astpPivotIn_active: Id {a6c9c124-5de5-4532-ac28-30489e3bb2bb}
   Action _astpPivotIn_entry: Id {a8fa57d0-3478-4e33-a7fb-56e0a3fc5e42}
   Action _astpPivotOut_active: Id {1b5a5545-2cbc-4640-8ac1-ee3d6846e106}
   Action _astpPivotOut_entry: Id {453454eb-9bde-4bd4-a989-f790d0fcd2d1}
   Action _astpRetract_Gui1_active: Id {9c1e0aee-7778-4a8f-a083-dae1dcfe84f4}
   Action _astpRetract_Gui1_entry: Id {cd6d199b-38de-45c2-8d32-91572ae3ce57}
   Action _astpRetract_Pous2_active: Id {6a9895eb-b600-43b7-8716-0d8072c24daa}
   Action _astpRetract_Pous2_entry: Id {295358fc-d4fe-4201-96ad-a1c1c70f6d60}
   Action stpCycle_Megagenial_active: Id {f41558d6-b881-4947-8649-a53b5a957e0e}
   Action stpDrop_Rail1_active: Id {4a9d4d90-45fb-4d7d-aad0-afa0f297d2d4}
   Action stpHoming_Active: Id {af655b4e-aa21-49ae-80b0-b983e3e6a8f9}
   Action stpHoming_Rail1_active: Id {56d49874-ad0c-400a-932d-c09aa003556e}
   Action stpHoming_Rail2_active: Id {05de02ac-fc4f-4dfa-bf73-dd333619d594}
   Action stpHoming_Rail3_active: Id {a8079511-f2ba-46af-a200-391749389f5a}
   Action stpHoming_Rail4_active: Id {1a90254e-196a-43a6-a57f-623383978a9d}
   Action stpInit_active: Id {10aa273c-50f4-48b2-827b-3d0220d77be7}
   Action stpInit_exit: Id {dcce3caa-9028-4c2f-8708-fd9c7506d3f5} *)
